// SIMATIC S7-200 project (STEP 7-Micro/WIN), CPU 224XP REL 02.01

SYMBOL_TABLE USUARIO1
P_PEATONES       I0.0
C_VERDE          Q0.0
C_AMBAR          Q0.1
C_ROJO           Q0.2
P_VERDE          Q0.3
P_ROJO           Q0.4
AUXILIAR         Q2.0
SEGURIDAD        Q2.1
END_SYMBOL_TABLE

SYMBOL_TABLE Símbolos S7-200
Primer_ciclo_ON  SM0.1    // ON sólo en el primer ciclo
END_SYMBOL_TABLE

ORGANIZATION_BLOCK PRINCIPAL:OB1
TITLE=COMENTARIOS DEL PROGRAMA
BEGIN
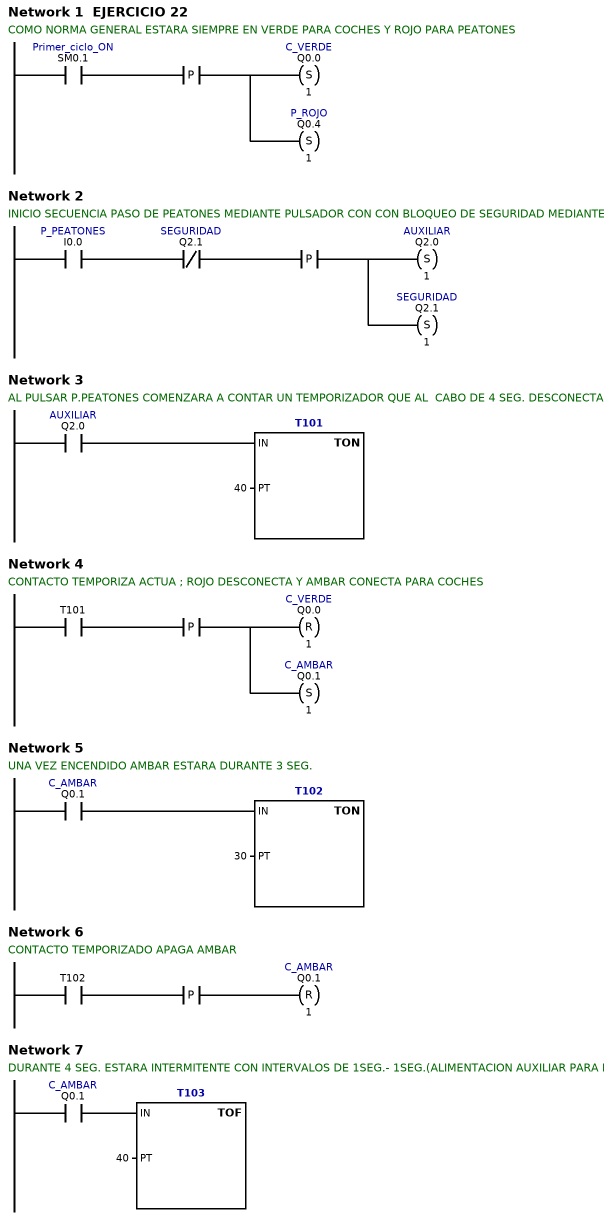
Network 1 // EJERCICIO 22
// COMO NORMA GENERAL ESTARA SIEMPRE EN VERDE PARA COCHES Y ROJO PARA PEATONES
LD     Primer_ciclo_ON:SM0.1
EU
S      C_VERDE:Q0.0, 1
S      P_ROJO:Q0.4, 1
Network 2
// INICIO SECUENCIA PASO DE PEATONES MEDIANTE PULSADOR CON CON BLOQUEO DE SEGURIDAD MEDIANTE MARCA AUXILIAR
// (network saved uncompiled; LAD cells follow)
// row 0: c0 -| |- P_PEATONES:I0.0  c1 -|/|- SEGURIDAD:Q2.1  c2 -|P|-  v  c3 -(S) AUXILIAR:Q2.0, 1
// row 1: c2 ^  c3 -(S) SEGURIDAD:Q2.1, 1
Network 3
// AL PULSAR P.PEATONES COMENZARA A CONTAR UN TEMPORIZADOR QUE AL  CABO DE 4 SEG. DESCONECTA VERDE COCHES Y CONECTA AMBAR
// (network saved uncompiled; LAD cells follow)
// row 0: c0 -| |- AUXILIAR:Q2.0  c1 --  c2 [TON T101 IN:=power@row0, PT:=40]
// row 1: c2 [box]
Network 4
// CONTACTO TEMPORIZA ACTUA ; ROJO DESCONECTA Y AMBAR CONECTA PARA COCHES
LD     T101
EU
R      C_VERDE:Q0.0, 1
S      C_AMBAR:Q0.1, 1
Network 5
// UNA VEZ ENCENDIDO AMBAR ESTARA DURANTE 3 SEG.
LD     C_AMBAR:Q0.1
TON    T102, 30
Network 6
// CONTACTO TEMPORIZADO APAGA AMBAR
LD     T102
EU
R      C_AMBAR:Q0.1, 1
Network 7
// DURANTE 4 SEG. ESTARA INTERMITENTE CON INTERVALOS DE 1SEG.- 1SEG.(ALIMENTACION AUXILIAR PARA EJECUCION DE ITERMITENCIA)
// (network saved uncompiled; LAD cells follow)
// row 0: c0 -| |- C_AMBAR:Q0.1  c1 [TOF T103 IN:=power@row0, PT:=40]
// row 1: c1 [box]
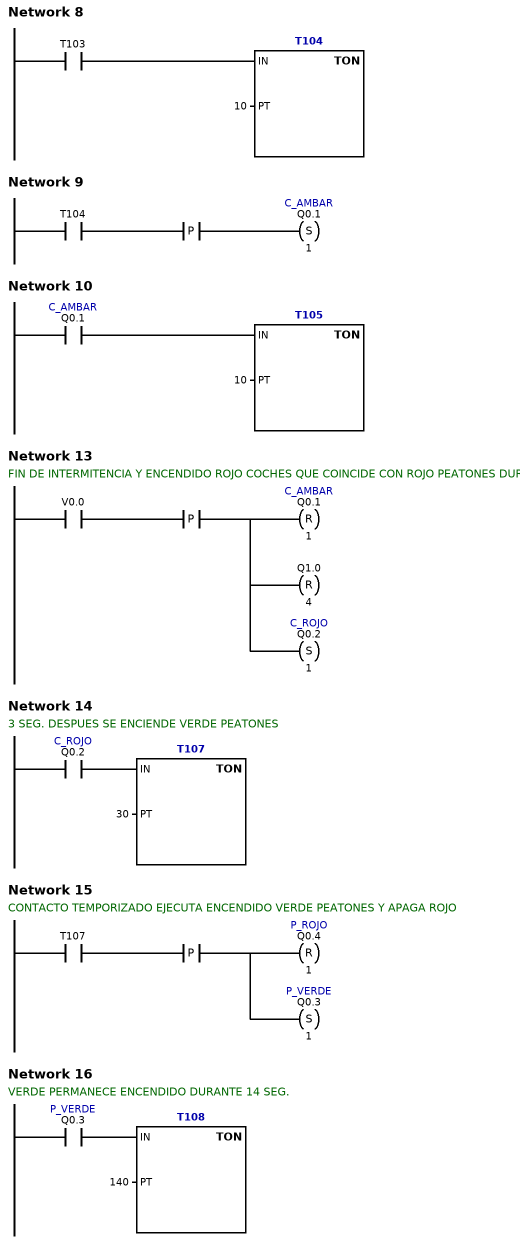
Network 8
// (network saved uncompiled; LAD cells follow)
// row 0: c0 -| |- T103  c1 --  c2 [TON T104 IN:=power@row0, PT:=10]
// row 1: c2 [box]
Network 9
// (network saved uncompiled; LAD cells follow)
// row 0: c0 -| |- T104  c1 -|P|-  c2 -(S) C_AMBAR:Q0.1, 1
Network 10
// (network saved uncompiled; LAD cells follow)
// row 0: c0 -| |- C_AMBAR:Q0.1  c1 --  c2 [TON T105 IN:=power@row0, PT:=10]
// row 1: c2 [box]
Network 13
// FIN DE INTERMITENCIA Y ENCENDIDO ROJO COCHES QUE COINCIDE CON ROJO PEATONES DURANTE 3 SEG.
// (network saved uncompiled; LAD cells follow)
// row 0: c0 -| |- V0.0  c1 -|P|-  v  c2 -(R) C_AMBAR:Q0.1, 1
// row 1: c1 ^v  c2 -(R) Q1.0, 4
// row 2: c1 ^  c2 -(S) C_ROJO:Q0.2, 1
Network 14
// 3 SEG. DESPUES SE ENCIENDE VERDE PEATONES 
// (network saved uncompiled; LAD cells follow)
// row 0: c0 -| |- C_ROJO:Q0.2  c1 [TON T107 IN:=power@row0, PT:=30]
// row 1: c1 [box]
Network 15
// CONTACTO TEMPORIZADO EJECUTA ENCENDIDO VERDE PEATONES Y APAGA ROJO
// (network saved uncompiled; LAD cells follow)
// row 0: c0 -| |- T107  c1 -|P|-  v  c2 -(R) P_ROJO:Q0.4, 1
// row 1: c1 ^  c2 -(S) P_VERDE:Q0.3, 1
Network 16
// VERDE PERMANECE ENCENDIDO DURANTE 14 SEG. 
// (network saved uncompiled; LAD cells follow)
// row 0: c0 -| |- P_VERDE:Q0.3  c1 [TON T108 IN:=power@row0, PT:=140]
// row 1: c1 [box]
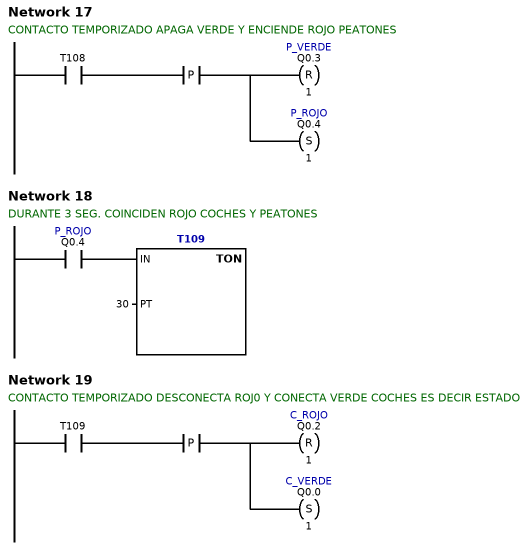
Network 17
// CONTACTO TEMPORIZADO APAGA VERDE Y ENCIENDE ROJO PEATONES
// (network saved uncompiled; LAD cells follow)
// row 0: c0 -| |- T108  c1 -|P|-  v  c2 -(R) P_VERDE:Q0.3, 1
// row 1: c1 ^  c2 -(S) P_ROJO:Q0.4, 1
Network 18
// DURANTE 3 SEG. COINCIDEN ROJO COCHES Y PEATONES 
// (network saved uncompiled; LAD cells follow)
// row 0: c0 -| |- P_ROJO:Q0.4  c1 [TON T109 IN:=power@row0, PT:=30]
// row 1: c1 [box]
Network 19
// CONTACTO TEMPORIZADO DESCONECTA ROJ0 Y CONECTA VERDE COCHES ES DECIR ESTADO INICIAL
// (network saved uncompiled; LAD cells follow)
// row 0: c0 -| |- T109  c1 -|P|-  v  c2 -(R) C_ROJO:Q0.2, 1
// row 1: c1 ^  c2 -(S) C_VERDE:Q0.0, 1
END_ORGANIZATION_BLOCK
